TYPE ST_PopUp_ToHmi :
STRUCT
	bVisible		: BOOL;
	nSymbol			: INT; //E_PopupSymbol;
	stText			: ST_Text;
	bButton01		: BOOL := TRUE;
	stButton01		: ST_HMI_BUTTON_OUT;
	bButton02		: BOOL := TRUE;
	stButton02		: ST_HMI_BUTTON_OUT;
	bButton03		: BOOL := TRUE;
	stButton03		: ST_HMI_BUTTON_OUT;
	bButton04		: BOOL := TRUE;
	stButton04		: ST_HMI_BUTTON_OUT;
END_STRUCT
END_TYPE

(* stored: Version 1.1.0.1, ProductVersion 3.1.4024.11
   DUT ST_PopUp_ToHmi: Id {997b9390-2d5a-4fcf-8398-ead4975fffe3} *)
